(* PLC project prj, KAIST_DSLAB noNameNow 1, author bwkim *)
(* stored: creationDateTime 2015-7-21T04:51:58, modificationDateTime 2015-7-21T04:51:58 *)

PROGRAM program2____sub1
  VAR
    FR_PTRIP_TON : null;
  END_VAR
  VAR
    FR_TRIP_TON : null;
  END_VAR
  VAR_OUTPUT
    PTRIP : BOOL := FALSE;
  END_VAR
  VAR_OUTPUT
    TRIP : BOOL := FALSE;
  END_VAR
  VAR_IN_OUT
    TRIP_LOGIC : BOOL := FALSE;
  END_VAR
  VAR_IN_OUT
    PTRIP_LOGIC : BOOL := FALSE;
  END_VAR
  VAR  (* added by the conversion: wires and edge detectors of the diagram *)
    _SEL_BOOL49_OUT : BOOL;
    _SEL_BOOL51_OUT : BOOL;
    _SEL_REAL52_OUT : ANY;
    _AND2_BOOL36_OUT : BOOL;
    _SEL_REAL50_OUT : ANY;
    _AND2_BOOL38_OUT : BOOL;
    _AND2_BOOL42_OUT : ANY;
  END_VAR

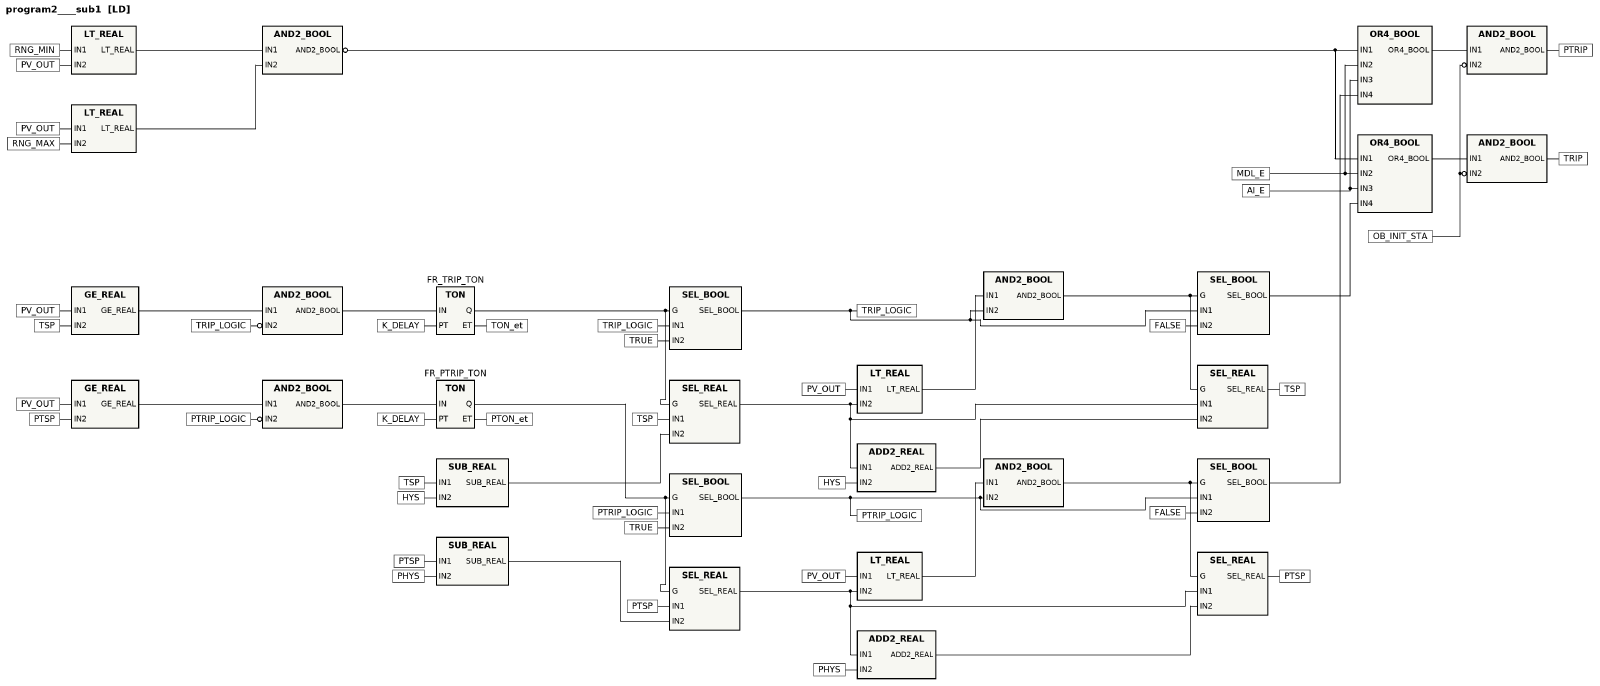
(* LD diagram, written out as Structured Text *)
FR_PTRIP_TON(IN := AND2_BOOL(GE_REAL(PV_OUT, PTSP), NOT PTRIP_LOGIC), PT := K_DELAY);
_SEL_BOOL49_OUT := SEL_BOOL(FR_PTRIP_TON.Q, PTRIP_LOGIC, TRUE);
PTRIP_LOGIC := _SEL_BOOL49_OUT;
PTON_et := FR_PTRIP_TON.ET;
FR_TRIP_TON(IN := AND2_BOOL(GE_REAL(PV_OUT, TSP), NOT TRIP_LOGIC), PT := K_DELAY);
_SEL_BOOL51_OUT := SEL_BOOL(FR_TRIP_TON.Q, TRIP_LOGIC, TRUE);
TRIP_LOGIC := _SEL_BOOL51_OUT;
TON_et := FR_TRIP_TON.ET;
_SEL_REAL52_OUT := SEL_REAL(FR_TRIP_TON.Q, TSP, SUB_REAL(TSP, HYS));
_AND2_BOOL36_OUT := AND2_BOOL(LT_REAL(PV_OUT, _SEL_REAL52_OUT), _SEL_BOOL51_OUT);
TSP := SEL_REAL(_AND2_BOOL36_OUT, _SEL_REAL52_OUT, ADD2_REAL(_SEL_REAL52_OUT, HYS));
_SEL_REAL50_OUT := SEL_REAL(FR_PTRIP_TON.Q, PTSP, SUB_REAL(PTSP, PHYS));
_AND2_BOOL38_OUT := AND2_BOOL(LT_REAL(PV_OUT, _SEL_REAL50_OUT), _SEL_BOOL49_OUT);
PTSP := SEL_REAL(_AND2_BOOL38_OUT, _SEL_REAL50_OUT, ADD2_REAL(_SEL_REAL50_OUT, PHYS));
_AND2_BOOL42_OUT := AND2_BOOL(LT_REAL(RNG_MIN, PV_OUT), LT_REAL(PV_OUT, RNG_MAX));
PTRIP := AND2_BOOL(OR4_BOOL(_AND2_BOOL42_OUT, MDL_E, AI_E, SEL_BOOL(_AND2_BOOL38_OUT, _SEL_BOOL49_OUT, FALSE)), NOT OB_INIT_STA);
TRIP := AND2_BOOL(OR4_BOOL(_AND2_BOOL42_OUT, MDL_E, AI_E, SEL_BOOL(_AND2_BOOL36_OUT, _SEL_BOOL51_OUT, FALSE)), NOT OB_INIT_STA);
END_PROGRAM
